FUNCTION_BLOCK OUT_ANY (* Data output to TextField *)
  (* Standard: 61499-1; Classification: GUI *)
  (* Version 0.1, 2002-05-03, JHC, Rockwell Automation, Made QI IV=true. *)
  (* Version 0.0, 2001-05-31, JHC, Rockwell Automation *)
  (* Compiler header: package fb.rt.hmi; *)
  (* Compiler Java IBM VisualAge 3.0 *)
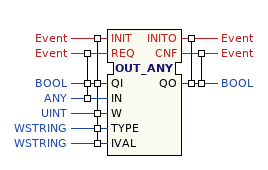
  EVENT_INPUT
    INIT WITH QI, W, TYPE, IVAL; (* Initialization *)
    REQ WITH QI, IN; (* Request *)
  END_EVENT
  EVENT_OUTPUT
    INITO WITH QO; (* Initialization Confirm *)
    CNF WITH QO; (* Service Confirmation *)
  END_EVENT
  VAR_INPUT
    QI : BOOL := true; (* Input event qualifier *)
    IN : ANY; (* Output value to convert *)
    W : UINT := 10; (* TextField width in chars *)
    TYPE : WSTRING := "ANY"; (* Data type name *)
    IVAL : WSTRING; (* Initial value *)
  END_VAR
  VAR_OUTPUT
    QO : BOOL; (* Output event qualifier *)
  END_VAR
  SERVICE OUT_ANY/TextField
    SEQUENCE normal_initialization
      OUT_ANY.INIT+(IVAL) -> TextField.initialize(IVAL) -> OUT_ANY.INITO+();
    END_SEQUENCE
    SEQUENCE initialization_inhibited
      OUT_ANY.INIT-() -> OUT_ANY.INITO-();
    END_SEQUENCE
    SEQUENCE normal_data_transfer
      OUT_ANY.REQ+(IN) -> TextField.setText(IN) -> OUT_ANY.CNF+();
    END_SEQUENCE
    SEQUENCE data_transfer_inhibited
      OUT_ANY.REQ-() -> OUT_ANY.CNF-();
    END_SEQUENCE
  END_SERVICE
END_FUNCTION_BLOCK
